FUNCTION_BLOCK FB_MixingValve EXTENDS FB_ActorContinous
VAR_INPUT
	nControlModeAutomatic : E_MixingValveControlMode; //control mode: 0 = position mode, 1 = heating mode, 2 = cooling mode
	fTemperatureExternal : REAL; //External temperature in °C
END_VAR
VAR_OUTPUT
END_VAR
VAR	
	{attribute 'OPC.UA.DA' := '1'}
	localSetParameters : ST_MixingValveSetParameters;
	
	//default parameters
	localDefaultParameters : ST_MixingValveDefaultParameters;	

	//analog converters for 0 - 10 V i/o signals
	InputConverter : FB_AnalogInput(fLowerLimit := 0, fUpperLimit := 90);
	OutputConverter : FB_AnalogOutput(fLowerLimit := 0, fUpperLimit := 100);
	
	//I/O Links
	nSetPoint_OUT		AT %Q* : INT; //Set position linked to terminal
	nOperatingPoint_IN 	AT %I* : INT; //Actual valve position linked to terminal
	
	//internal variables
	nControlMode			: E_MixingValveControlMode;	
	fSetPoint_internal 		: REAL; //internal, control mode depending setpoint between 0.0 and 100.0
	
	//controllers
	PI_Controller_Heating		: FB_CTRL_PI;
	PI_Controller_Cooling		: FB_CTRL_PI;
	PI_Controler_Parameters 	: ST_CTRL_PI_PARAMS;
	
END_VAR

MAIN();
SelectValveControlMode();
ControlValve();

METHOD ControlValve : BOOL
VAR_INPUT
END_VAR
VAR
END_VAR
//set control parameters
PI_Controler_Parameters.fKp 			:= localDefaultParameters.fControlerAmplification;
PI_Controler_Parameters.tTn 			:= DINT_TO_TIME(localDefaultParameters.fControlerIntegralTime);
PI_Controler_Parameters.fOutMaxLimit	:= 100.0;
PI_Controler_Parameters.fOutMinLimit	:= 0.0;
PI_Controler_Parameters.tTaskCycleTime	:= GlobalVariables.tTaskCycleTime;
PI_Controler_Parameters.tCtrlCycleTime	:= DINT_TO_TIME(500);
PI_Controler_Parameters.bARWOnIPartOnly	:= TRUE;

IF bSetStatusOn THEN
	CASE nControlMode OF
		0: //position mode
		fSetPoint_internal := fSetPoint;
		
		1: //heating mode
		PI_Controller_Heating (
				fSetpointValue	:= fSetPoint,
				fActualValue	:= fTemperatureExternal,
				fManSyncValue	:= 0,
				bSync			:= FALSE,
				eMode			:= 2, (* mode active *)
				bHold			:= FALSE,
				stParams		:= PI_Controler_Parameters);
		fSetPoint_internal := LREAL_TO_REAL(PI_Controller_Heating.fOut);
				
		2: //cooling mode
		PI_Controller_Cooling (
			fSetpointValue	:= fTemperatureExternal,
			fActualValue	:= fSetPoint,
			fManSyncValue	:= 0,
			bSync			:= FALSE,
			eMode			:= 2, (* mode active *)
			bHold			:= FALSE,
			stParams		:= PI_Controler_Parameters);
		fSetPoint_internal := LREAL_TO_REAL(PI_Controller_Cooling.fOut);
	END_CASE
ELSE
	fSetPoint_internal := localDefaultParameters.fDefaultPosition;
END_IF
END_METHOD

METHOD SelectValveControlMode : BOOL
VAR_INPUT
END_VAR
IF control.bManualModeActivated THEN
	nControlMode := localSetParameters.nControlModeManual;
ELSIF control.bAlgorithmModeActivated AND bAlgorithmPermission THEN
	nControlMode := localSetParameters.nControlModeAlgorithm;
ELSE
	nControlMode := nControlModeAutomatic;
END_IF
END_METHOD

METHOD PROTECTED  SetSetPointLimits : BOOL
VAR_INPUT
END_VAR
CASE nControlMode OF
	0: //position mode
	aSetPointLimits := localDefaultParameters.aSetPointLimitsPosition;

	1: //heating mode
	aSetPointLimits := localDefaultParameters.aSetPointLimitsTemperature;
	
	2: //cooling mode
	aSetPointLimits := localDefaultParameters.aSetPointLimitsTemperature;
END_CASE
END_METHOD

METHOD SetState_AI_AO : BOOL
VAR
END_VAR
//setpoint and control state
setPointState.fSetPoint := fSetPoint;
CASE nControlMode OF
	0: //position mode
	setPointState.sSetPointUnit := 'percent';
	
	1: //heating mode
	setPointState.sSetPointUnit := 'degreeC';
	
	2: //cooling mode
	setPointState.sSetPointUnit := 'degreeC';
END_CASE

IF localDefaultParameters.bFeedbackSignal = TRUE THEN //Set operating point if there is a feedback signal 
	InputConverter(nValue := nOperatingPoint_IN);
	setPointState.fOperatingPoint := InputConverter.fValue;
	setPointState.sOperatingPointUnit := 'percent';
	setPointState.aSetPointLimits := aSetPointLimits;
	IF setPointState.fOperatingPoint > 0 THEN //Set control state if valve is open
		controlState.bStatusOn := TRUE;
	ELSE
		controlState.bStatusOn := FALSE;
	END_IF
END_IF;

//Output
OutputConverter(fValue := fSetPoint_internal);
nSetPoint_OUT := OutputConverter.nValue;  //converts real setpoint for terminal
END_METHOD

PROPERTY ST_DefaultParameters : REFERENCE TO ST_MixingValveDefaultParameters
SET
localDefaultParameters := ST_DefaultParameters;
END_SET
END_PROPERTY

END_FUNCTION_BLOCK

(* stored: Version 1.1.0.1, ProductVersion 3.1.4024.9
   POU FB_MixingValve: Id {60dbc338-d028-4fcc-a2a7-9fe749ce4d3c}, SpecialFunc None
   Method ControlValve: Id {1e52182a-8bdc-49bd-b2bd-13ceeb4d93b8}
   Method SelectValveControlMode: Id {69d2db34-6658-4b13-ae91-6cb6bcdc3229}
   Method SetSetPointLimits: Id {a8c83337-88ad-4b4d-a894-cec3559c40a9}
   Method SetState_AI_AO: Id {be832a62-70d4-4ec0-8ee4-578237454401}
   Property ST_DefaultParameters: Id {1a42851e-de6a-48b1-b7bd-13b0312684ce}
   Set Set: Id {a86ebf94-4f5d-419b-bd12-1e8c85044a39} *)
